FUNCTION Call_ADSCommunication

RF_Data_Ready(CLK := instVisionSensorConveyor.Finished);

IF RF_Data_Ready.Q THEN
	Detected_Material := instVisionSensorConveyor.Parttype;
	Data_Ready := TRUE;
END_IF

END_FUNCTION

(* stored: Version 1.1.0.1
   POU Call_ADSCommunication: Id {6a0c7f72-4ce4-4ca7-9795-4028d2ce8ab4}, SpecialFunc None *)
